Fanuc KAREL source: kb00196.KL

-- PROVISIONAL review KL for V940-1; original PC SHA256 785a3a75380dbf9819993c4452fd2c40913bb75fc54b02a2f0471365ae471b4f
-- Incomplete behavior may be omitted. Consult companion uncertainty JSON. Do not deploy.
PROGRAM KB00196
%NOLOCKGROUP
BEGIN
  -- V9_ZERO_TABLE_METADATA_HINT layout=0002_ascii; no indexed target words; source/name/runtime held
  -- UNRESOLVED_PC offsets 5-14; opcodes 3F,75
  -- UNRESOLVED_PC offsets 19-26; opcodes 9D,23
  -- UNRESOLVED_PC offsets 31-38; opcodes 9D,23
  -- UNRESOLVED_PC offsets 43-52; opcodes 3F,75
  -- UNRESOLVED_PC offsets 57-89; opcodes 27,22,2A,22,22,22,2A,31
  -- UNRESOLVED_PC offsets 94-98; opcodes 7F
END KB00196
